// TIA Portal V20 export
TYPE "type_emRelations_em0_cmStatus"
// stored: Access Published, Namespace Unit1
   STRUCT
      Stacker1NgBoxDetect : "LBC_typeDigitalSignalControlNode";
      Stacker1NgBoxFullDetect : "LBC_typeDigitalSignalControlNode";
      Stacker1NgBoxLoadingUpDown : "LBC_typeTwoWayActuatorControlNode";
      Stacker1NgBoxUnitMoverBwdFwd : "LBC_typeTwoWayActuatorControlNode";
      Stacker1NgBoxClampLeftOpenClose : "LBC_typeTwoWayActuatorControlNode";
      Stacker1NgBoxClampRightOpenClose : "LBC_typeTwoWayActuatorControlNode";
      Stacker1NgBoxClampMoverOpenClose : "LBC_typeTwoWayActuatorControlNode";
      Stacker1NgBoxLiftDownUp : "LBC_typeTwoWayActuatorControlNode";
      Stacker1NgBoxLockDownUp : "LBC_typeTwoWayActuatorControlNode";
   END_STRUCT;
   // // Stacker1NgBoxLoadingUpDown.commands.commandHomePos : STAKC #1 NG CLAMP Z-AXIS UP
   // // Stacker1NgBoxLoadingUpDown.commands.commandWorkPos : STAKC #1 NG CLAMP Z-AXIS DOWN
   // // Stacker1NgBoxUnitMoverBwdFwd.commands.commandHomePos : STAKC #1 NG CLAMP UNIT MOVER BACKWARD
   // // Stacker1NgBoxUnitMoverBwdFwd.commands.commandWorkPos : STAKC #1 NG CLAMP UNIT MOVER FORWARD
   // // Stacker1NgBoxClampLeftOpenClose.commands.commandHomePos : STACK #1 NG CLAMP LEFT OPEN
   // // Stacker1NgBoxClampLeftOpenClose.commands.commandWorkPos : STACK #1 NG CLAMP LEFT CLOSE
   // // Stacker1NgBoxClampRightOpenClose.commands.commandHomePos : STACK #1 NG CLAMP RIGHT OPEN
   // // Stacker1NgBoxClampRightOpenClose.commands.commandWorkPos : STACK #1 NG CLAMP RIGHT CLOSE
   // // Stacker1NgBoxLiftDownUp.commands.commandHomePos : STACK #1 NG BOX LIFT UP
   // // Stacker1NgBoxLiftDownUp.commands.commandWorkPos : STACK #1 NG BOX LIFT DOWN
   // // Stacker1NgBoxLockDownUp.commands.commandHomePos : STACK #1 NG BOX LOCK DOWN
   // // Stacker1NgBoxLockDownUp.commands.commandWorkPos : STACK #1 NG BOX LOCK UP
END_TYPE
